FUNCTION_BLOCK IN_TEXT_S (* STRING input from TextArea-see IN_TEXT *)
  (* Standard: 61499-1; Classification: GUI *)
  (* Version 0.2, 2002-05-03, JHC, Rockwell Automation, Made QI IV=true. *)
  (* Version 0.1, 2001-11-26, JHC, Rockwell Automation, Copied/Modified from IN_TEXT. *)
  (* Version 0.0, 2001-10-09, JHC, Rockwell Automation, Copied/Modified from IN_ANY *)
  (* Compiler header: package fb.rt.hmi.*; *)
  (* Compiler Java IBM VisualAge 3.0 *)
  (* Compiler Java IBM Jikes 1.0.6 *)
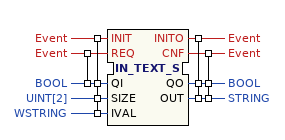
  EVENT_INPUT
    INIT WITH QI, SIZE, IVAL;
    REQ WITH QI;
  END_EVENT
  EVENT_OUTPUT
    INITO WITH QO, OUT;
    CNF WITH QO, OUT;
  END_EVENT
  VAR_INPUT
    QI : BOOL := true;
    SIZE : ARRAY [0..1] OF UINT := [10,50]; (* [rows,columns] *)
    IVAL : WSTRING;
  END_VAR
  VAR_OUTPUT
    QO : BOOL; (* 1=OK,0=Error *)
    OUT : STRING;
  END_VAR
END_FUNCTION_BLOCK
